TYPE ST_Erreur :
STRUCT
	xState:BOOL; 		//shows the current error state
	iId : INT; 			//error number currently active
	sMessage : STRING; 	//error message for the active error
END_STRUCT
END_TYPE

(* stored: Version 1.1.0.1, ProductVersion 3.1.4020.6
   DUT ST_Erreur: Id {dffce1a9-47c9-4b68-8fdc-b9291109262a} *)
